INTERFACE I_OrderedDictionaryTreeNode EXTENDS I_CollectionNode

METHOD PUBLIC Clone
VAR_INPUT
	Node : I_OrderedDictionaryTreeNode;
END_VAR
END_METHOD

PROPERTY PUBLIC Height : DINT
GET
END_GET
SET
END_SET
END_PROPERTY

PROPERTY PUBLIC Key : T_MAXSTRING
GET
END_GET
END_PROPERTY

PROPERTY PUBLIC Left : I_OrderedDictionaryTreeNode
GET
END_GET
SET
END_SET
END_PROPERTY

PROPERTY PUBLIC Next : I_OrderedDictionaryTreeNode
GET
END_GET
SET
END_SET
END_PROPERTY

PROPERTY PUBLIC NodeBufferPointer : Pointer To Byte
GET
END_GET
END_PROPERTY

PROPERTY PUBLIC NodeBufferSize : UDINT
GET
END_GET
END_PROPERTY

PROPERTY PUBLIC Previous : I_OrderedDictionaryTreeNode
GET
END_GET
SET
END_SET
END_PROPERTY

METHOD Reinitialize
VAR_INPUT
	Key : T_MAXSTRING;
	Source : ANY;
END_VAR
END_METHOD

PROPERTY PUBLIC Right : I_OrderedDictionaryTreeNode
GET
END_GET
SET
END_SET
END_PROPERTY

END_INTERFACE

(* stored: Version 1.1.0.1, ProductVersion 3.1.4024.12
   Itf I_OrderedDictionaryTreeNode: Id {429c1971-9387-4ece-a9e2-e3d2db0fbc73}
   Method Clone: Id {771df79c-7a3b-45f7-8b1e-b78167e8a9e0}
   Property Height: Id {dd295a66-fbd1-4637-87e1-20608bd534e8}
   Get Get: Id {5a560fad-5dbd-4fda-8a6d-845ef4bde448}
   Set Set: Id {caec95f5-7e22-4331-ac67-244d2c96cf86}
   Property Key: Id {f505aa6b-54da-4e9e-96ab-5c323e363448}
   Get Get: Id {20c5c0fe-3915-4784-950e-69c37a702cad}
   Property Left: Id {e9f3cb4f-f17e-4353-ab55-e1952fbeef92}
   Get Get: Id {fec4d1b0-abb4-429c-8d10-3458cdd49340}
   Set Set: Id {c0a1d3b9-d981-485d-b6bb-0e3103923fc2}
   Property Next: Id {4a100539-46a2-47aa-b4f2-2b88820570ad}
   Get Get: Id {a44078d8-32c7-4594-a273-72bda471d05c}
   Set Set: Id {8b11fd91-f0e0-45b5-91d2-af25d22d3016}
   Property NodeBufferPointer: Id {baa9f846-4833-4cbf-bcec-ce498040bc87}
   Get Get: Id {36ace33f-3f88-43c9-9dd2-3cf072d8d786}
   Property NodeBufferSize: Id {27d7a6ad-6864-4329-838d-11d422206d6c}
   Get Get: Id {3cc18e55-6f0d-4be1-8c44-d0b125135902}
   Property Previous: Id {992fdc46-792a-4eca-8a38-ff4f51dc16ed}
   Get Get: Id {cd2d9738-286a-45cc-981a-de67e73da7d1}
   Set Set: Id {5a405ae4-9c1d-4cbb-b818-b5b6b9f7f8a3}
   Method Reinitialize: Id {15835b1d-1819-4226-851f-15303db91a25}
   Property Right: Id {0d14ff1a-4f17-4925-867a-c80334e8af02}
   Get Get: Id {a659acee-d960-41d4-8616-512ab533594d}
   Set Set: Id {dad0992a-6cb9-40c0-b629-b698b81f8649} *)
